// Mitsubishi GX Works2 project: 20151022   PLC: Q03UDV

PROGRAM P1
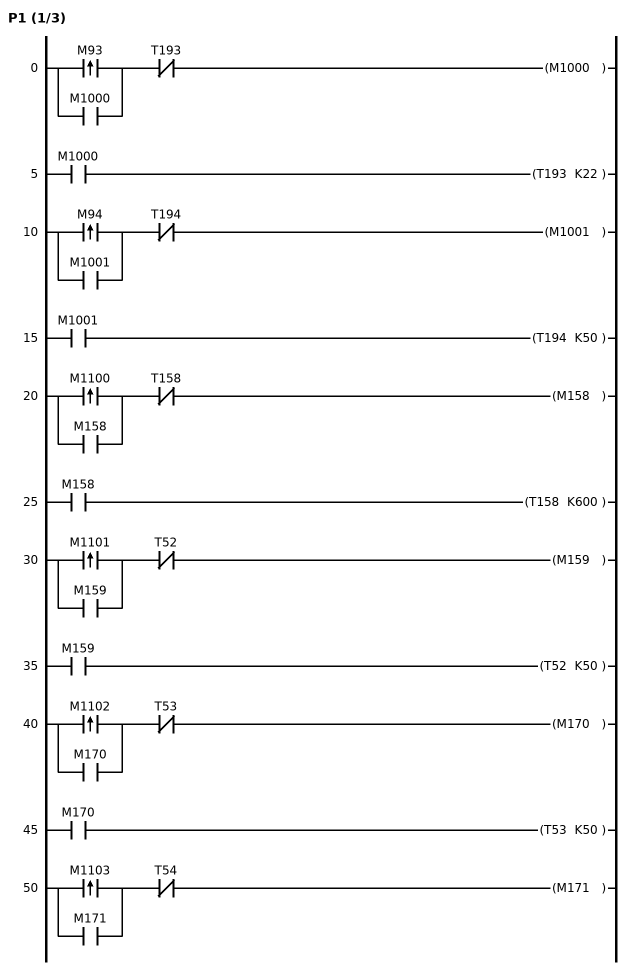
0     LDP     M93
      OR      M1000
      ANI     T193
      OUT     M1000
5     LD      M1000
      OUT     T193 K22
10    LDP     M94
      OR      M1001
      ANI     T194
      OUT     M1001
15    LD      M1001
      OUT     T194 K50
20    LDP     M1100
      OR      M158
      ANI     T158
      OUT     M158
25    LD      M158
      OUT     T158 K600
30    LDP     M1101
      OR      M159
      ANI     T52
      OUT     M159
35    LD      M159
      OUT     T52 K50
40    LDP     M1102
      OR      M170
      ANI     T53
      OUT     M170
45    LD      M170
      OUT     T53 K50
50    LDP     M1103
      OR      M171
      ANI     T54
      OUT     M171
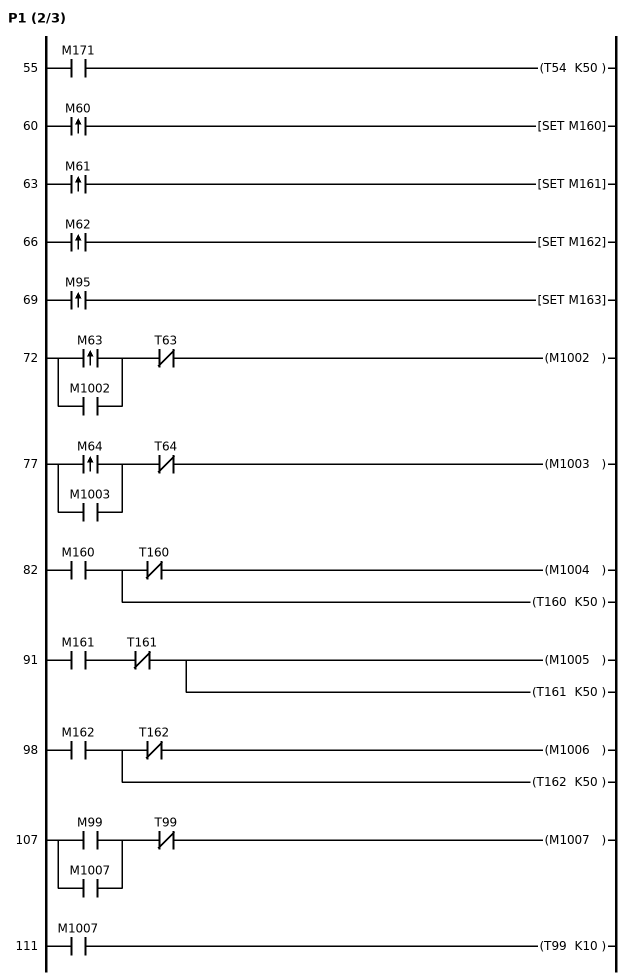
55    LD      M171
      OUT     T54 K50
60    LDP     M60
      SET     M160
63    LDP     M61
      SET     M161
66    LDP     M62
      SET     M162
69    LDP     M95
      SET     M163
72    LDP     M63
      OR      M1002
      ANI     T63
      OUT     M1002
77    LDP     M64
      OR      M1003
      ANI     T64
      OUT     M1003
82    LD      M160
      MPS
      ANI     T160
      OUT     M1004
      MPP
      OUT     T160 K50
91    LD      M161
      ANI     T161
      OUT     M1005
      OUT     T161 K50
98    LD      M162
      MPS
      ANI     T162
      OUT     M1006
      MPP
      OUT     T162 K50
107   LD      M99
      OR      M1007
      ANI     T99
      OUT     M1007
111   LD      M1007
      OUT     T99 K10
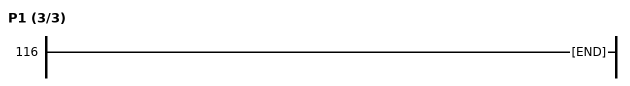
116   END
END_PROGRAM

PROGRAM P2
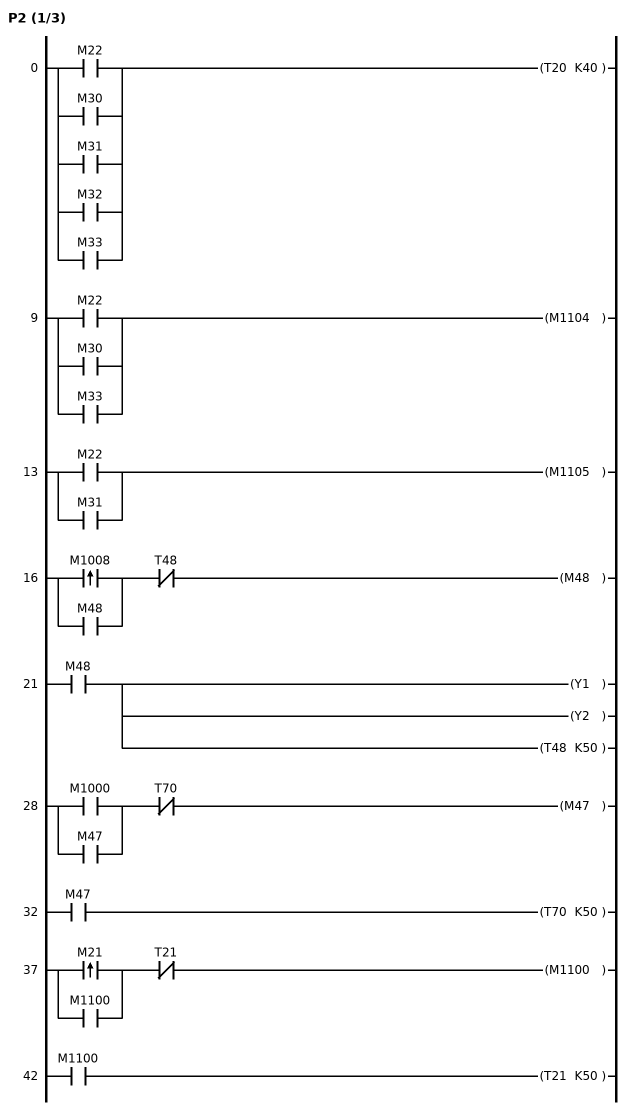
0     LD      M22
      OR      M30
      OR      M31
      OR      M32
      OR      M33
      OUT     T20 K40
9     LD      M22
      OR      M30
      OR      M33
      OUT     M1104
13    LD      M22
      OR      M31
      OUT     M1105
16    LDP     M1008
      OR      M48
      ANI     T48
      OUT     M48
21    LD      M48
      OUT     Y1
      OUT     Y2
      OUT     T48 K50
28    LD      M1000
      OR      M47
      ANI     T70
      OUT     M47
32    LD      M47
      OUT     T70 K50
37    LDP     M21
      OR      M1100
      ANI     T21
      OUT     M1100
42    LD      M1100
      OUT     T21 K50
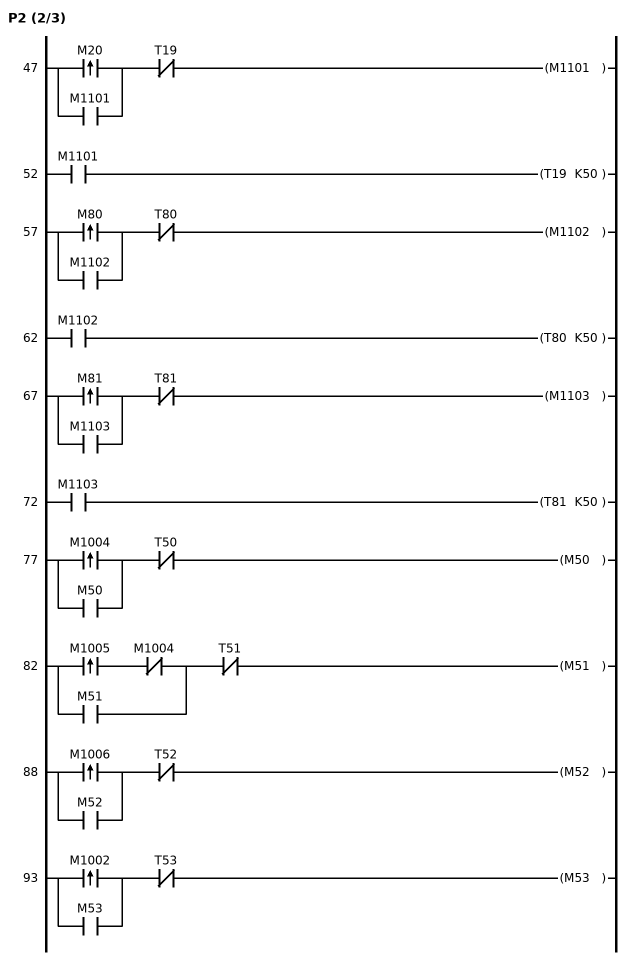
47    LDP     M20
      OR      M1101
      ANI     T19
      OUT     M1101
52    LD      M1101
      OUT     T19 K50
57    LDP     M80
      OR      M1102
      ANI     T80
      OUT     M1102
62    LD      M1102
      OUT     T80 K50
67    LDP     M81
      OR      M1103
      ANI     T81
      OUT     M1103
72    LD      M1103
      OUT     T81 K50
77    LDP     M1004
      OR      M50
      ANI     T50
      OUT     M50
82    LDP     M1005
      ANI     M1004
      OR      M51
      ANI     T51
      OUT     M51
88    LDP     M1006
      OR      M52
      ANI     T52
      OUT     M52
93    LDP     M1002
      OR      M53
      ANI     T53
      OUT     M53
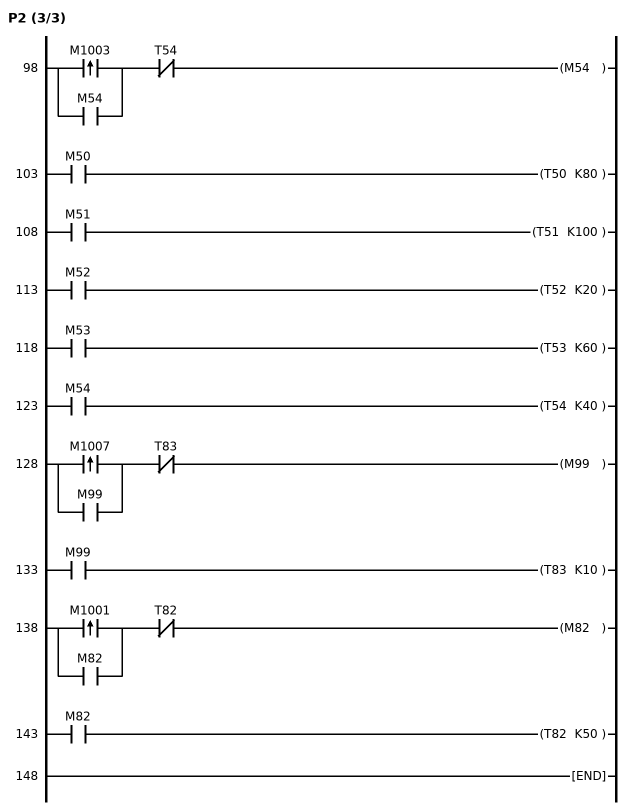
98    LDP     M1003
      OR      M54
      ANI     T54
      OUT     M54
103   LD      M50
      OUT     T50 K80
108   LD      M51
      OUT     T51 K100
113   LD      M52
      OUT     T52 K20
118   LD      M53
      OUT     T53 K60
123   LD      M54
      OUT     T54 K40
128   LDP     M1007
      OR      M99
      ANI     T83
      OUT     M99
133   LD      M99
      OUT     T83 K10
138   LDP     M1001
      OR      M82
      ANI     T82
      OUT     M82
143   LD      M82
      OUT     T82 K50
148   END
END_PROGRAM
